// TIA Portal V20 export
DATA_BLOCK "PM01"   // DB207
// stored: MemoryReserve 100
   VAR
      "AIRS01 UNWINDER LEFT AIR SHAFT ON" : Bool;
      SPARE_1 : Bool;
      "AIRS02 UNWINDER RIGHT AIR SHAFT ON" : Bool;
      SPARE_2 : Bool;
      SPARE_3 : Bool;
      SPARE_4 : Bool;
      SPARE_5 : Bool;
      SPARE_6 : Bool;
      "C03 UNWINDER SUPPORT UNIT TRANSFER FORWARD" : Bool;
      "C03 UNWINDER SUPPORT UNIT TRANSFER BACKWARD" : Bool;
      "C04 ELECTRODE SHAFT SUPPORTER UP" : Bool;
      "C04 ELECTRODE SHAFT SUPPORTER DOWN" : Bool;
      SPARE_7 : Bool;
      SPARE_8 : Bool;
      SPARE_9 : Bool;
      SPARE_10 : Bool;
   END_VAR
BEGIN
END_DATA_BLOCK
